SUBAPPLICATION Uebung_019 (* Umschalten einer Maske *)
  (* Standard: 61499-2; Description: Copyright (c) 2023 Meisterschulen am Ostbahnhof This program and the accompanying materials are made available under the terms of the Eclipse Public License 2.0 which is available at https://www.eclipse.org/legal/epl-2.0/ SPDX-License-Identifier: EPL-2.0 *)
  (* Version 1.0, 2023-10-23, Franz Höpfinger, Meisterschulen am Ostbahnhof, initial API and implementation and/or initial documentation *)
  PACKAGE Uebungen;
  IMPORT Uebungen::const::UT::DefaultPool::DataMask_M1;
  IMPORT Uebungen::const::UT::DefaultPool::DataMask_M2;
  IMPORT logiBUS::io::DI::logiBUS_DI::Input_I1;
  IMPORT logiBUS::io::DI::logiBUS_DI::Input_I2;
  IMPORT logiBUS::io::DI::logiBUS_DI_Events::BUTTON_SINGLE_CLICK;
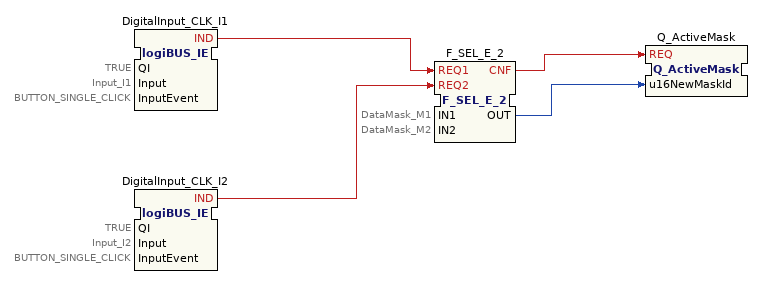
  FBS
    DigitalInput_CLK_I1 : logiBUS::io::DI::logiBUS_IE(QI := TRUE, Input := Input_I1, InputEvent := BUTTON_SINGLE_CLICK);
    Q_ActiveMask : isobus::UT::Q::Q_ActiveMask;
    DigitalInput_CLK_I2 : logiBUS::io::DI::logiBUS_IE(QI := TRUE, Input := Input_I2, InputEvent := BUTTON_SINGLE_CLICK);
    F_SEL_E_2 : eclipse4diac::utils::selection::F_SEL_E_2(IN1 := DataMask_M1, IN2 := DataMask_M2);
  END_FBS
  EVENT_CONNECTIONS
    DigitalInput_CLK_I1.IND TO F_SEL_E_2.REQ1;
    DigitalInput_CLK_I2.IND TO F_SEL_E_2.REQ2;
    F_SEL_E_2.CNF TO Q_ActiveMask.REQ;
  END_CONNECTIONS
  DATA_CONNECTIONS
    F_SEL_E_2.OUT TO Q_ActiveMask.u16NewMaskId;
  END_CONNECTIONS
END_SUBAPPLICATION
